// TIA Portal V19 program export: 6 tag tables, 0 data types, 4 data blocks, 10 code blocks (in call order from the OBs), 11 instance data blocks

VAR_GLOBAL   // PLC tag table "Default tag table"
   RETVAL_WWW AT %MW80 : Int;
   LampeStart AT %Q1.0 : Bool;
   Start_Stop AT %M10.0 : Bool;
   Compteur AT %MW2 : Int;
   PieceMax AT %MW100 : Int;
   "Compteur Bonnes Pièces" AT %MW10 : Int;
   "Compteur Mauvaises Pièces" AT %MW12 : Int;
   "Pointeur 1" AT %MD50 : DWord;
   "Pointeur 2" AT %MD54 : DWord;
   "A CHANGER" AT %MW200 : Word;
END_VAR

VAR_GLOBAL   // PLC tag table "Entrées"
   PART_AV AT %I0.0 : Bool;   // Détection pièce disponible
   B2 AT %I0.1 : Bool;   // Détection pièces (pas noir)
   B4 AT %I0.2 : Bool;   // Barrière sécurité
   "1B1" AT %I0.4 : Bool;   // Vérin 1A1 position haute
   "1B2" AT %I0.5 : Bool;   // Vérin 1A1 position basse
   "2B1" AT %I0.6 : Bool;   // Vérin 2A1 rentré
   Start AT %I1.0 : Bool;   // Départ cycle
   Stop AT %I1.1 : Bool;   // Fin cycle
   Reset AT %I1.3 : Bool;   // Initialisation station
   Analogique AT %IW800 : Int;   // Capteur analogique
END_VAR

VAR_GLOBAL   // PLC tag table "Mémoires"
   "Hauteur (pourcentage)" AT %MD0 : Real;   // Valeur de la hauteur de la pièce en pourcentage
   "Activer Q1" AT %M4.0 : Bool;   // Mémoire pour activer Q1
   "Mémoire compteur noires" AT %M4.1 : Bool;   // Mémoire pour les fronts montants du cpt noires
   "Mémoire compteur mauvaise hauteur" AT %M4.2 : Bool;   // Mémoire pour les fronts montants du cpt mauvaises pièces
   "Mémoire compteur bonne hauteur" AT %M4.3 : Bool;   // Mémoire pour les fronts montants du cpt bonnes pièces
   "Clock 1Hz" AT %M250.5 : Bool;
   "Clock 2Hz" AT %M250.3 : Bool;
   "Clock 0,625Hz" AT %M250.6 : Bool;
   "Clock 0,5Hz" AT %M250.7 : Bool;
   "Clock 1,5Hz" AT %M250.4 : Bool;
   "Clock 2,5Hz" AT %M250.2 : Bool;
   "Clock 5Hz" AT %M250.1 : Bool;
   "Clock 10Hz" AT %M250.0 : Bool;
   RETVAL_WWW AT %MW80 : Int;
   Start_Stop AT %M10.0 : Bool;
   Compteur AT %MW2 : Int;
   PieceMax AT %MW100 : Int;
   "Compteur Bonnes Pièces" AT %MW10 : Int;
   "Compteur Mauvaises Pièces" AT %MW12 : Int;
   "Pointeur 1" AT %MD50 : DWord;
   "Pointeur 2" AT %MD54 : DWord;
   "A CHANGER" AT %MW200 : Word;
   "NB Bonnes Pièces" AT %MW26 : Word;   // Nombre des bonnes pièces à afficher sur le web serveur
   "NB Mauvaises Pièces" AT %MW28 : Word;   // Nombre des mauvaises pièces à afficher sur le web serveur
END_VAR

VAR_GLOBAL   // PLC tag table "Sorties"
   "1M2" AT %Q0.0 : Bool;   // Descente vérin élévation pièce
   "1M1" AT %Q0.1 : Bool;   // Montée vérin élévation pièce
   "2M1" AT %Q0.2 : Bool;   // Sortie vérin éjection pièce
   "3M1" AT %Q0.3 : Bool;   // Activation toboggan pneumatique
   LStart AT %Q1.0 : Bool;   // Lampe BP Start
   LReset AT %Q1.1 : Bool;   // Lampe BP Reset
   Q1 AT %Q1.2 : Bool;   // Voyant lumineux Q1
   Q2 AT %Q1.3 : Bool;   // Voyant lumineux Q2
END_VAR

VAR_GLOBAL   // PLC tag table "Test - Copy"
   test1 AT %M120.0 : Bool;
   test2 AT %M120.1 : Bool;
END_VAR

VAR_GLOBAL   // PLC tag table "Test"
   test1 AT %M120.0 : Bool;
   test2 AT %M120.1 : Bool;
END_VAR

DATA_BLOCK "DB Bonnes Pièces"   // DB14
// stored: AutoNumber false
   VAR RETAIN
      "Nb_J-1" : Int;
      "Nb_J-2" : Int;
      "Nb_J-3" : Int;
      "Nb_J-4" : Int;
      "Nb_J-5" : Int;
      "Nb_J-6" : Int;
      "Nb_J-7" : Int;
      "Nb_J-8" : Int;
      "Nb_J-9" : Int;
      "Nb_J-10" : Int;
      "Nb_J-11" : Int;
      "Nb_J-12" : Int;
      "Nb_J-13" : Int;
      "Nb_J-14" : Int;
      "Nb_J-15" : Int;
      "Nb_J-16" : Int;
      "Nb_J-17" : Int;
      "Nb_J-18" : Int;
      "Nb_J-19" : Int;
      "Nb_J-20" : Int;
      "Nb_J-21" : Int;
      "Nb_J-22" : Int;
      "Nb_J-23" : Int;
      "Nb_J-24" : Int;
      "Nb_J-25" : Int;
      "Nb_J-26" : Int;
      "Nb_J-27" : Int;
      "Nb_J-28" : Int;
      "Nb_J-29" : Int;
      "Nb_J-30" : Int;
      "Nb_J-31" : Int;
   END_VAR
BEGIN
END_DATA_BLOCK

DATA_BLOCK "DB Mauvaises Pièces"   // DB13
// stored: AutoNumber false
   VAR RETAIN
      "Nb_J-1" : Int;
      "Nb_J-2" : Int;
      "Nb_J-3" : Int;
      "Nb_J-4" : Int;
      "Nb_J-5" : Int;
      "Nb_J-6" : Int;
      "Nb_J-7" : Int;
      "Nb_J-8" : Int;
      "Nb_J-9" : Int;
      "Nb_J-10" : Int;
      "Nb_J-11" : Int;
      "Nb_J-12" : Int;
      "Nb_J-13" : Int;
      "Nb_J-14" : Int;
      "Nb_J-15" : Int;
      "Nb_J-16" : Int;
      "Nb_J-17" : Int;
      "Nb_J-18" : Int;
      "Nb_J-19" : Int;
      "Nb_J-20" : Int;
      "Nb_J-21" : Int;
      "Nb_J-22" : Int;
      "Nb_J-23" : Int;
      "Nb_J-24" : Int;
      "Nb_J-25" : Int;
      "Nb_J-26" : Int;
      "Nb_J-27" : Int;
      "Nb_J-28" : Int;
      "Nb_J-29" : Int;
      "Nb_J-30" : Int;
      "Nb_J-31" : Int;
   END_VAR
BEGIN
END_DATA_BLOCK

DATA_BLOCK "Grosse data"   // DB1
   VAR RETAIN
      "Grosse donnée" : Bool;
      "Une autre grosse donnée" : Int;
   END_VAR
BEGIN
END_DATA_BLOCK

DATA_BLOCK "Mémoires"   // DB2
   VAR RETAIN
      "Mode Manuel" : Bool;
      "Affichage hauteur" : Int;
      "HMI BP Ascenceur Haut" : Bool;
      "HMI BP Ascenceur Bas" : Bool;
      "HMI BP Ejection" : Bool;
      "HMI SW Glissière" : Bool;
      "Erreur Montée Ascenceur" : Int;
      "Erreur Descente Ascenceur" : Int;
      "Erreur Ejection" : Int;
      "Erreur Capteurs" : Int;
   END_VAR
BEGIN
END_DATA_BLOCK

ORGANIZATION_BLOCK "Main"   // OB1, LAD, ProgramCycle
TITLE = "Main Program Sweep (Cycle)"
   VAR_TEMP
      OB1_EV_CLASS : Byte;   // Bits 0-3 = 1 (Coming event), Bits 4-7 = 1 (Event class 1)
      OB1_SCAN_1 : Byte;   // 1 (Cold restart scan 1 of OB 1), 3 (Scan 2-n of OB 1)
      OB1_PRIORITY : Byte;   // Priority of OB Execution
      OB1_OB_NUMBR : Byte;   // 1 (Organization block 1, OB1)
      OB1_RESERVED_1 : Byte;   // Reserved for system
      OB1_RESERVED_2 : Byte;   // Reserved for system
      OB1_PREV_CYCLE : Int;   // Cycle time of previous OB1 scan (milliseconds)
      OB1_MIN_CYCLE : Int;   // Minimum cycle time of OB1 (milliseconds)
      OB1_MAX_CYCLE : Int;   // Maximum cycle time of OB1 (milliseconds)
      OB1_DATE_TIME : Date_And_Time;   // Date and time OB1 started
   END_VAR
BEGIN

REGION Network 1
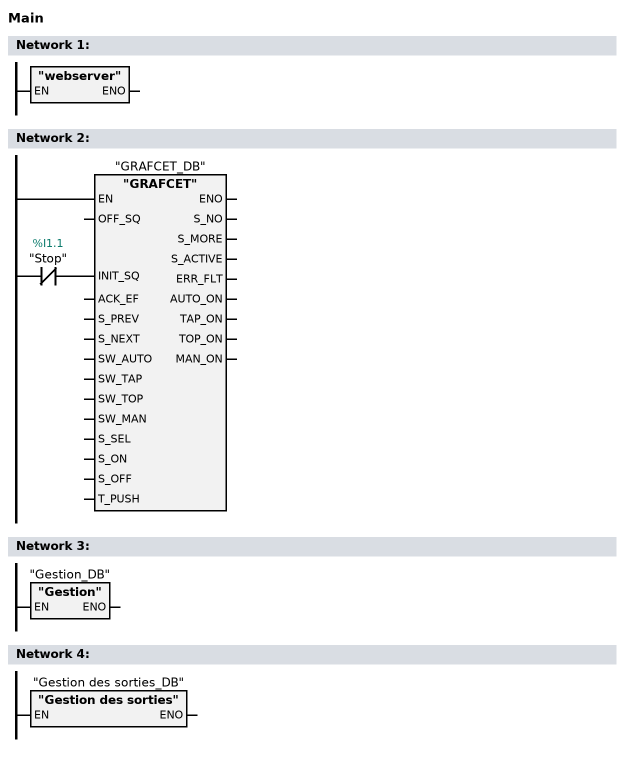
   RUNG wire#powerrail
      "webserver"()
   END_RUNG
   // the same network as SCL:
   "webserver"();
END_REGION

REGION Network 2
   RUNG wire#powerrail
      "GRAFCET_DB"(INIT_SQ := wire#w1, OFF_SQ :=, ACK_EF :=, S_PREV :=, S_NEXT :=, SW_AUTO :=, SW_TAP :=, SW_TOP :=, SW_MAN :=, S_SEL :=, S_ON :=, S_OFF :=, T_PUSH :=, S_NO =>, S_MORE =>, S_ACTIVE =>, ERR_FLT =>, AUTO_ON =>, TAP_ON =>, TOP_ON =>, MAN_ON =>)
   END_RUNG
   RUNG wire#powerrail
      I_Contact( "Stop" )
   END_RUNG wire#w1
   // the same network as SCL:
   "GRAFCET_DB"(INIT_SQ := NOT "Stop");   // "GRAFCET"
END_REGION

REGION Network 3
   RUNG wire#powerrail
      "Gestion_DB"()
   END_RUNG
   // the same network as SCL:
   "Gestion_DB"();   // "Gestion"
END_REGION

REGION Network 4
   RUNG wire#powerrail
      "Gestion des sorties_DB"()
   END_RUNG
   // the same network as SCL:
   "Gestion des sorties_DB"();   // "Gestion des sorties"
END_REGION

NETWORK
TITLE = Call system diagnostics block
      CALL  "RSE_FB", "RSE_DB";
END_ORGANIZATION_BLOCK

FUNCTION "webserver" : Void   // FC1, LAD
   VAR_TEMP
      RET_VAL_1 : Int;
   END_VAR
BEGIN

REGION Network 1
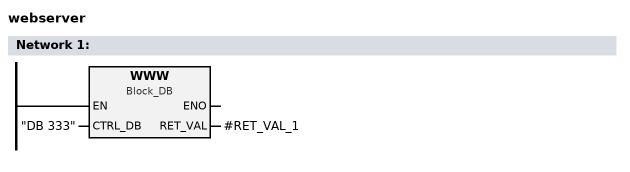
   RUNG wire#powerrail
      { S7_Templates := "value_type := Block_DB" } WWW(CTRL_DB := "DB 333", RET_VAL => #RET_VAL_1)
   END_RUNG
   // the same network as SCL:
   #RET_VAL_1 := WWW(CTRL_DB := "DB 333");
END_REGION
END_FUNCTION

FUNCTION_BLOCK "GRAFCET"   // FB1, GRAPH
   VAR_INPUT
      OFF_SQ { ExternalAccessible := 'False'; ExternalVisible := 'False'; ExternalWritable := 'False'} : Bool := false;   // Turn sequence off
      INIT_SQ { ExternalAccessible := 'False'; ExternalVisible := 'False'; ExternalWritable := 'False'} : Bool := false;   // Set sequence to initial state
      ACK_EF { ExternalAccessible := 'False'; ExternalVisible := 'False'; ExternalWritable := 'False'} : Bool := false;   // Acknowledge all errors and faults
      S_PREV { ExternalAccessible := 'False'; ExternalVisible := 'False'; ExternalWritable := 'False'} : Bool := false;   // Output previous step in parameter S_NO
      S_NEXT { ExternalAccessible := 'False'; ExternalVisible := 'False'; ExternalWritable := 'False'} : Bool := false;   // Indicate next step in parameter S_NO
      SW_AUTO { ExternalAccessible := 'False'; ExternalVisible := 'False'; ExternalWritable := 'False'} : Bool := false;   // Automatic mode
      SW_TAP { ExternalAccessible := 'False'; ExternalVisible := 'False'; ExternalWritable := 'False'} : Bool := false;   // Semiautomatic/switch with transition
      SW_TOP { ExternalAccessible := 'False'; ExternalVisible := 'False'; ExternalWritable := 'False'} : Bool := false;   // Semiautomatic/ignore transition
      SW_MAN { ExternalAccessible := 'False'; ExternalVisible := 'False'; ExternalWritable := 'False'} : Bool := false;   // Manual mode
      S_SEL { ExternalAccessible := 'False'; ExternalVisible := 'False'; ExternalWritable := 'False'} : Int := 0;   // Select step to be output to S_NO
      S_ON { ExternalAccessible := 'False'; ExternalVisible := 'False'; ExternalWritable := 'False'} : Bool := false;   // Activate step indicated in S_NO
      S_OFF { ExternalAccessible := 'False'; ExternalVisible := 'False'; ExternalWritable := 'False'} : Bool := false;   // Deactivate step indicated S_NO
      T_PUSH { ExternalAccessible := 'False'; ExternalVisible := 'False'; ExternalWritable := 'False'} : Bool := false;   // Enable transition to switch in semi automatic mode
   END_VAR
   VAR_OUTPUT
      S_NO { ExternalAccessible := 'False'; ExternalVisible := 'False'; ExternalWritable := 'False'} : Int := 0;   // Step number
      S_MORE { ExternalAccessible := 'False'; ExternalVisible := 'False'; ExternalWritable := 'False'} : Bool := false;   // More steps are available and can be shown in S_NO
      S_ACTIVE { ExternalAccessible := 'False'; ExternalVisible := 'False'; ExternalWritable := 'False'} : Bool := false;   // Step indicated in S_NO is active
      ERR_FLT { ExternalAccessible := 'False'; ExternalVisible := 'False'; ExternalWritable := 'False'} : Bool := false;   // Interlock or supervision group error
      AUTO_ON { ExternalAccessible := 'False'; ExternalVisible := 'False'; ExternalWritable := 'False'} : Bool := false;   // Automatic mode is active
      TAP_ON { ExternalAccessible := 'False'; ExternalVisible := 'False'; ExternalWritable := 'False'} : Bool := false;   // Semiautomatic mode/step with transition enabled
      TOP_ON { ExternalAccessible := 'False'; ExternalVisible := 'False'; ExternalWritable := 'False'} : Bool := false;   // Semiautomatic mode/ignore transition enabled
      MAN_ON { ExternalAccessible := 'False'; ExternalVisible := 'False'; ExternalWritable := 'False'} : Bool := false;   // Manual mode is active
   END_VAR
   VAR
      S_DISPLAY { ExternalAccessible := 'False'; ExternalVisible := 'False'; ExternalWritable := 'False'} : Int;   // Internal display of output parameter S_NO
      S_SEL_OLD { ExternalAccessible := 'False'; ExternalVisible := 'False'; ExternalWritable := 'False'} : Int;   // Previous value in S_SEL
      S_DISPIDX { ExternalAccessible := 'False'; ExternalVisible := 'False'; ExternalWritable := 'False'} : Byte;   // Index of the step in S_NO
      T_DISPIDX { ExternalAccessible := 'False'; ExternalVisible := 'False'; ExternalWritable := 'False'} : Byte;   // Index of the transition displayed in T_NO
      MOP { ExternalAccessible := 'False'; ExternalVisible := 'False'; ExternalWritable := 'False'} : Struct   // Mode
         AUTO : Bool := true;   // Status: automatic mode
         MAN : Bool := false;   // Status: manual mode
         TAP : Bool := false;   // Status: semi automatic/switch with transition
         TOP : Bool := false;   // Status: semi automatic/ignore transition
         ACK_S : Bool := false;   // Request: acknowledge step at parameter S_NO
         REG_S : Bool := false;   // Request: register step indicated in S_NO
         T_PREV : Bool := false;   // Request: output previous valid transition in T_NO
         T_NEXT : Bool := false;   // Request: output next valid transition in T_NO
         LOCK : Bool := true;   // Status: interlocks activated
         SUP : Bool := true;   // Status: supervisions activated
         ACKREQ : Bool := true;   // Status: acknowledgment required
         SSKIP : Bool := false;   // Status: "Skip steps" enabled
         OFF : Bool := false;   // Request: deactivate all steps
         INIT : Bool := true;   // Request: set sequence to initial state
         HALT : Bool := false;   // Status: sequence halted
         TMS_HALT : Bool := false;   // Status: all internal timers held
         OPS_ZERO : Bool := false;   // Status: set all operands processed with N, L, D instructions to 0
         SACT_DISP : Bool := true;   // Status: display active steps only
         SEF_DISP : Bool := false;   // Status: display only steps with errors and disrupted steps
         SALL_DISP : Bool := false;   // Status: display all steps
         S_PREV : Bool := false;   // Request: output previous step to S_NO
         S_NEXT : Bool := false;   // Request: Output next step at S_NO parameter
         S_SELOK : Bool := false;   // Request: output step number from S_SEL to S_NO
         S_ON : Bool := false;   // Request: activate step indicated in S_NO
         S_OFF : Bool := false;   // Request: deactivate step at parameter S_NO
         T_PUSH : Bool := false;   // Request: transition switching enabled
         REG : Bool := false;   // Request: register all interlock and supervision errors
         ACK : Bool := false;   // Request: acknowledge all interlock and supervision errors
         IL_PERM : Bool := false;   // Status: permanent processing of all interlocks
         T_PERM : Bool := false;   // Status: permanent processing of all transitions
         ILP_MAN : Bool := false;   // Status: permanent processing of all interlocks in manual mode
      END_STRUCT;
      TICKS { ExternalAccessible := 'False'; ExternalVisible := 'False'; ExternalWritable := 'False'} : Struct   // Clock speeds
         DELTA : Time := T#0ms;   // Time difference between cycles
         OLD : Time := T#0ms;   // 10 ms clock counter value in last cycle
         NEW : Time := T#0ms;   // 10 ms clock counter value in this cycle
      END_STRUCT;
      SQ_FLAGS { ExternalAccessible := 'False'; ExternalVisible := 'False'; ExternalWritable := 'False'} : Struct   // Sequence bit memory
         ERR_FLT : Bool := false;   // Interlock and supervision group error
         ERROR : Bool := false;   // Interlock group error
         FAULT : Bool := false;   // Supervision group error
         RT_FAIL : Bool := false;   // Runtime error
         NO_SNO : Bool := false;   // Requested step number not found
         NF_OFL : Bool := false;   // Overflow: too many ON or OFF requests
         SA_OFL : Bool := false;   // Overflow: too many steps active
         TV_OFL : Bool := false;   // Overflow: too many valid transitions
         MSG_OFL : Bool := false;   // Overflow: not enough system resources for ALARM_S
         NO_SWI : Bool := false;   // Do not switch in this cycle
         CYC_OP : Bool := false;   // Cyclic execution of the sequence after initialization
         AS_MSG : Bool := true;   // Alarms during runtime enabled or disabled by instruction
         AS_SEND : Bool := false;   // Send alarms from WR_USMSG or only enter in diagnostics buffer
         SQ_BUSY : Bool := false;   // Internal edge bit memory for sequence processing
         SA_BUSY : Bool := false;   // Internal edge bit memory for sequence processing
         AS_SIG : Bool := false;   // Edge bit memory for alarms from Alarm_S and Alarm_SQ
      END_STRUCT;
   END_VAR
BEGIN
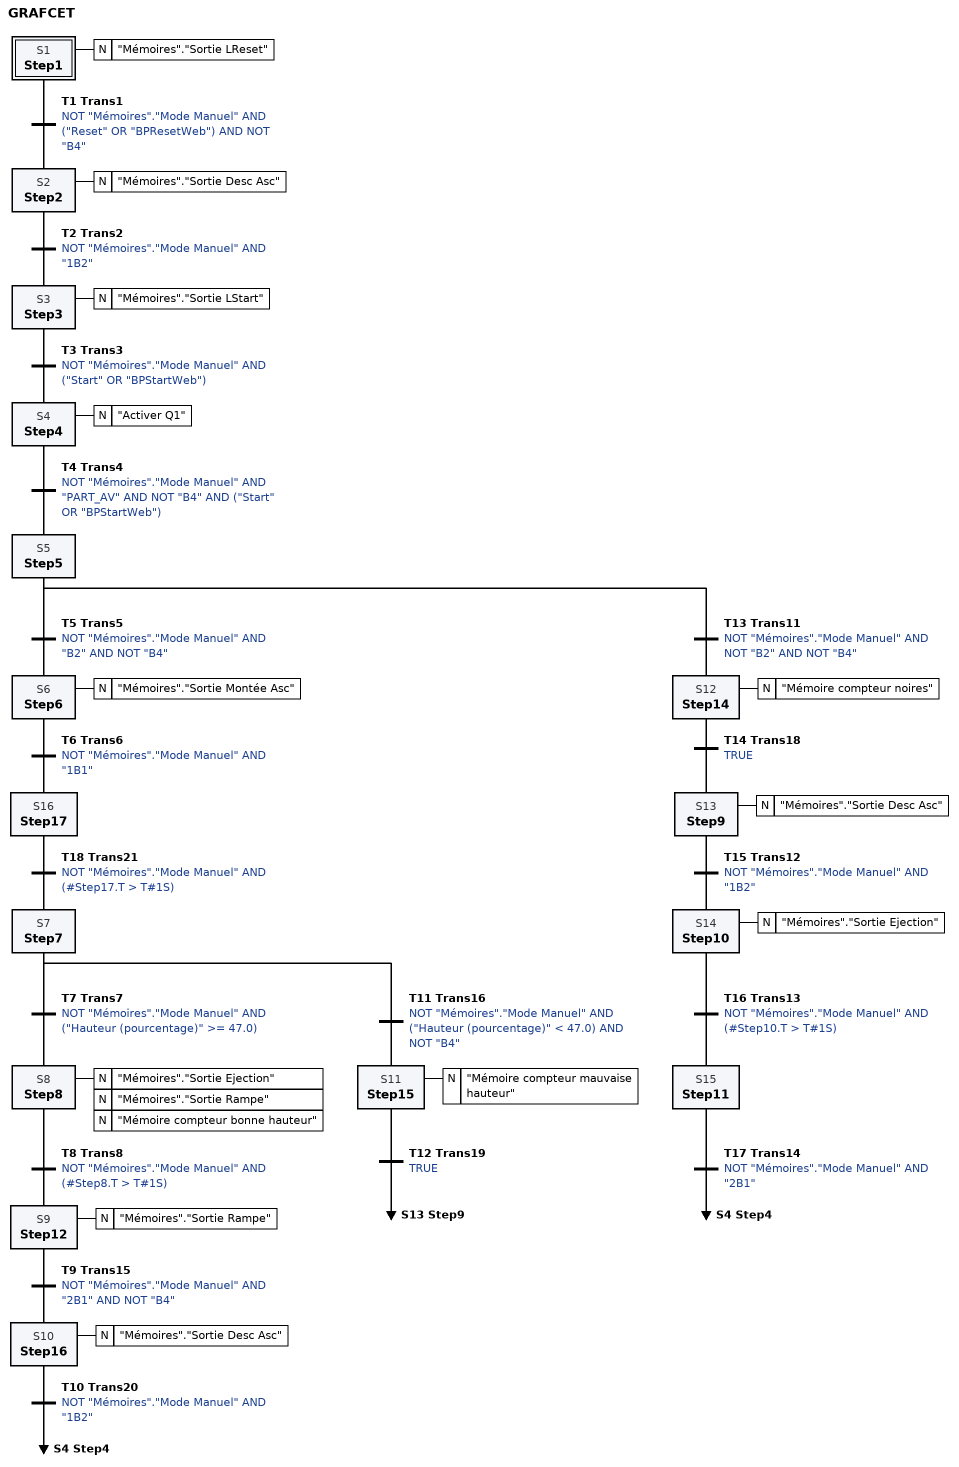
   // sequencer 1: GRAFCET de la séquence de tri
   INITIAL_STEP Step1:   // S1
              N    "Mémoires"."Sortie LReset"
   END_STEP
   TRANSITION Trans1 FROM Step1 TO Step2   // T1
      := NOT "Mémoires"."Mode Manuel" AND ("Reset" OR "BPResetWeb") AND NOT "B4";
   END_TRANSITION
   STEP Step2:   // S2
              N    "Mémoires"."Sortie Desc Asc"
   END_STEP
   TRANSITION Trans2 FROM Step2 TO Step3   // T2
      := NOT "Mémoires"."Mode Manuel" AND "1B2";
   END_TRANSITION
   STEP Step3:   // S3
              N    "Mémoires"."Sortie LStart"
   END_STEP
   TRANSITION Trans3 FROM Step3 TO Step4   // T3
      := NOT "Mémoires"."Mode Manuel" AND ("Start" OR "BPStartWeb");
   END_TRANSITION
   STEP Step4:   // S4
              N    "Activer Q1"
   END_STEP
   TRANSITION Trans4 FROM Step4 TO Step5   // T4
      := NOT "Mémoires"."Mode Manuel" AND "PART_AV" AND NOT "B4" AND ("Start" OR "BPStartWeb");
   END_TRANSITION
   STEP Step5:   // S5
   END_STEP
   TRANSITION Trans5 FROM Step5 TO Step6   // T5
      := NOT "Mémoires"."Mode Manuel" AND "B2" AND NOT "B4";
   END_TRANSITION
   TRANSITION Trans11 FROM Step5 TO Step14   // T13
      := NOT "Mémoires"."Mode Manuel" AND NOT "B2" AND NOT "B4";
   END_TRANSITION
   STEP Step6:   // S6
              N    "Mémoires"."Sortie Montée Asc"
   END_STEP
   TRANSITION Trans6 FROM Step6 TO Step17   // T6
      := NOT "Mémoires"."Mode Manuel" AND "1B1";
   END_TRANSITION
   STEP Step7:   // S7
   END_STEP
   TRANSITION Trans7 FROM Step7 TO Step8   // T7
      := NOT "Mémoires"."Mode Manuel" AND ("Hauteur (pourcentage)" >= 47.0);
   END_TRANSITION
   TRANSITION Trans16 FROM Step7 TO Step15   // T11
      := NOT "Mémoires"."Mode Manuel" AND ("Hauteur (pourcentage)" < 47.0) AND NOT "B4";
   END_TRANSITION
   STEP Step8:   // S8
              N    "Mémoires"."Sortie Ejection"
              N    "Mémoires"."Sortie Rampe"
              N    "Mémoire compteur bonne hauteur"
   END_STEP
   TRANSITION Trans8 FROM Step8 TO Step12   // T8
      := NOT "Mémoires"."Mode Manuel" AND (#Step8.T > T#1S);
   END_TRANSITION
   STEP Step9:   // S13
              N    "Mémoires"."Sortie Desc Asc"
   END_STEP
   TRANSITION Trans12 FROM Step9 TO Step10   // T15
      := NOT "Mémoires"."Mode Manuel" AND "1B2";
   END_TRANSITION
   STEP Step10:   // S14
              N    "Mémoires"."Sortie Ejection"
   END_STEP
   TRANSITION Trans13 FROM Step10 TO Step11   // T16
      := NOT "Mémoires"."Mode Manuel" AND (#Step10.T > T#1S);
   END_TRANSITION
   STEP Step11:   // S15
   END_STEP
   TRANSITION Trans14 FROM Step11 TO Step4   // T17, jump
      := NOT "Mémoires"."Mode Manuel" AND "2B1";
   END_TRANSITION
   STEP Step12:   // S9
              N    "Mémoires"."Sortie Rampe"
   END_STEP
   TRANSITION Trans15 FROM Step12 TO Step16   // T9
      := NOT "Mémoires"."Mode Manuel" AND "2B1" AND NOT "B4";
   END_TRANSITION
   STEP Step14:   // S12
              N    "Mémoire compteur noires"
   END_STEP
   TRANSITION Trans18 FROM Step14 TO Step9   // T14
      := TRUE;
   END_TRANSITION
   STEP Step15:   // S11
              N    "Mémoire compteur mauvaise hauteur"
   END_STEP
   TRANSITION Trans19 FROM Step15 TO Step9   // T12, jump
      := TRUE;
   END_TRANSITION
   STEP Step16:   // S10
              N    "Mémoires"."Sortie Desc Asc"
   END_STEP
   TRANSITION Trans20 FROM Step16 TO Step4   // T10, jump
      := NOT "Mémoires"."Mode Manuel" AND "1B2";
   END_TRANSITION
   STEP Step17:   // S16
   END_STEP
   TRANSITION Trans21 FROM Step17 TO Step7   // T18
      := NOT "Mémoires"."Mode Manuel" AND (#Step17.T > T#1S);
   END_TRANSITION
END_FUNCTION_BLOCK

FUNCTION_BLOCK "Gestion"   // FB2, LAD
   VAR
      "Code erreur" : Word;
      "FM Noires" : Bool;
      "FM Mauvaises" : Bool;
      "FM Bonnes" : Bool;
   END_VAR
   VAR_TEMP   // added for the SCL form of the ladder/FBD networks
      _w1 : Bool;
   END_VAR
BEGIN

REGION Network 1: Scale de la valeur d'entrée analogique
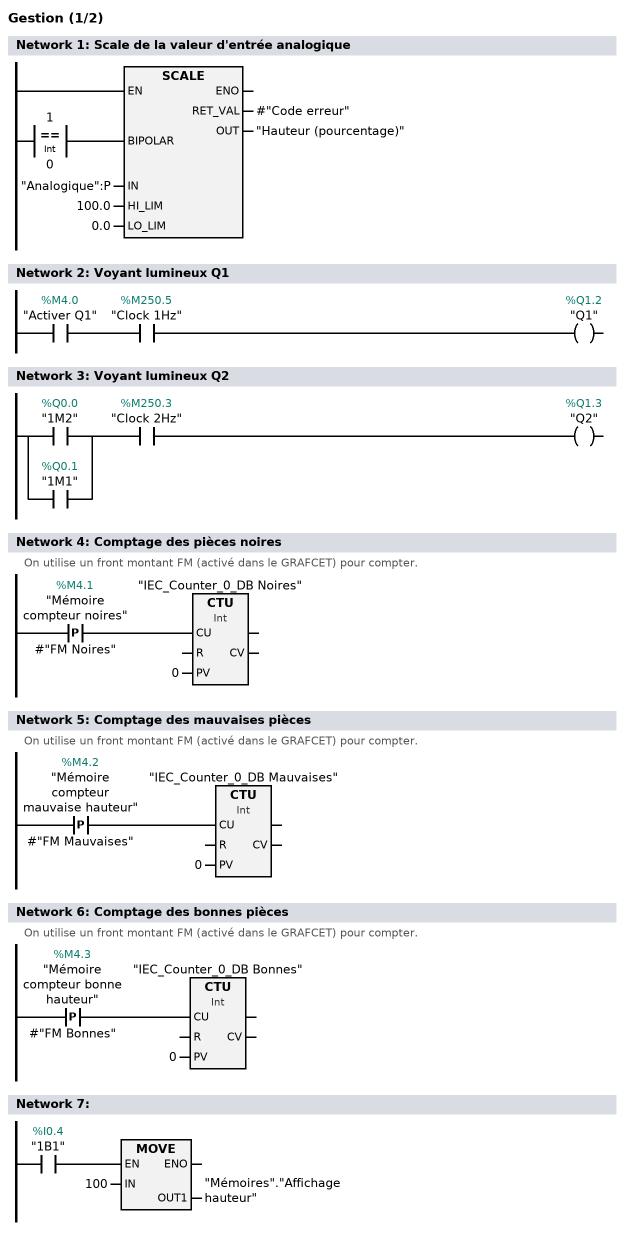
   #"Code erreur" := SCALE(BIPOLAR := 1 = 0,
                           IN := "Analogique":P,
                           HI_LIM := 100.0,
                           LO_LIM := 0.0,
                           OUT => "Hauteur (pourcentage)");
END_REGION

REGION Network 2: Voyant lumineux Q1
   RUNG wire#powerrail
      Contact( "Activer Q1" )
      Contact( "Clock 1Hz" )
      Coil( "Q1" )
   END_RUNG
   // the same network as SCL:
   "Q1" := "Activer Q1" AND "Clock 1Hz";
END_REGION

REGION Network 3: Voyant lumineux Q2
   RUNG wire#powerrail
      Contact( "1M2" )
      wire#w1
      Contact( "Clock 2Hz" )
      Coil( "Q2" )
   END_RUNG
   RUNG wire#powerrail
      Contact( "1M1" )
   END_RUNG wire#w1
   // the same network as SCL:
   "Q2" := ("1M2" OR "1M1") AND "Clock 2Hz";
END_REGION

REGION Network 4: Comptage des pièces noires
   // On utilise un front montant FM (activé dans le GRAFCET) pour compter.
   RUNG wire#powerrail
      P_Contact(operand := "Mémoire compteur noires", bit := #"FM Noires")
      { S7_Templates := "value_type := Int" } "IEC_Counter_0_DB Noires".CTU(r :=, pv := 0, cv =>)
   END_RUNG
   // the same network as SCL:
   #_w1 := "Mémoire compteur noires" AND NOT #"FM Noires";   // rising edge of "Mémoire compteur noires"
   #"FM Noires" := "Mémoire compteur noires";
   "IEC_Counter_0_DB Noires".CTU(CU := #_w1, PV := 0);
END_REGION

REGION Network 5: Comptage des mauvaises pièces
   // On utilise un front montant FM (activé dans le GRAFCET) pour compter.
   RUNG wire#powerrail
      P_Contact(operand := "Mémoire compteur mauvaise hauteur", bit := #"FM Mauvaises")
      { S7_Templates := "value_type := Int" } "IEC_Counter_0_DB Mauvaises".CTU(r :=, pv := 0, cv =>)
   END_RUNG
   // the same network as SCL:
   #_w1 := "Mémoire compteur mauvaise hauteur" AND NOT #"FM Mauvaises";   // rising edge of "Mémoire compteur mauvaise hauteur"
   #"FM Mauvaises" := "Mémoire compteur mauvaise hauteur";
   "IEC_Counter_0_DB Mauvaises".CTU(CU := #_w1, PV := 0);
END_REGION

REGION Network 6: Comptage des bonnes pièces
   // On utilise un front montant FM (activé dans le GRAFCET) pour compter.
   RUNG wire#powerrail
      P_Contact(operand := "Mémoire compteur bonne hauteur", bit := #"FM Bonnes")
      { S7_Templates := "value_type := Int" } "IEC_Counter_0_DB Bonnes".CTU(r :=, pv := 0, cv =>)
   END_RUNG
   // the same network as SCL:
   #_w1 := "Mémoire compteur bonne hauteur" AND NOT #"FM Bonnes";   // rising edge of "Mémoire compteur bonne hauteur"
   #"FM Bonnes" := "Mémoire compteur bonne hauteur";
   "IEC_Counter_0_DB Bonnes".CTU(CU := #_w1, PV := 0);
END_REGION

REGION Network 7
   RUNG wire#powerrail
      Contact( "1B1" )
      { S7_GenerateENO := "TRUE" } Move(in := 100, out1 => "Mémoires"."Affichage hauteur")
   END_RUNG
   // the same network as SCL:
   IF "1B1" THEN "Mémoires"."Affichage hauteur" := 100; END_IF;
END_REGION

REGION Network 8
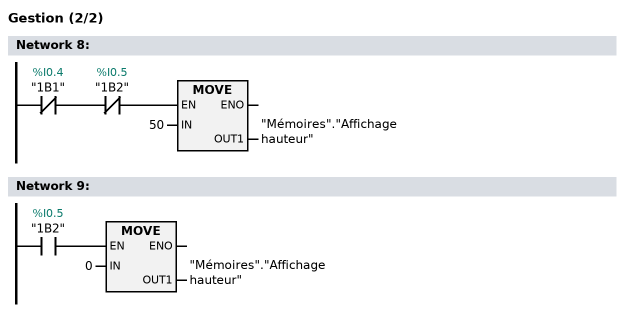
   RUNG wire#powerrail
      I_Contact( "1B1" )
      I_Contact( "1B2" )
      { S7_GenerateENO := "TRUE" } Move(in := 50, out1 => "Mémoires"."Affichage hauteur")
   END_RUNG
   // the same network as SCL:
   IF NOT "1B1" AND NOT "1B2" THEN "Mémoires"."Affichage hauteur" := 50; END_IF;
END_REGION

REGION Network 9
   RUNG wire#powerrail
      Contact( "1B2" )
      { S7_GenerateENO := "TRUE" } Move(in := 0, out1 => "Mémoires"."Affichage hauteur")
   END_RUNG
   // the same network as SCL:
   IF "1B2" THEN "Mémoires"."Affichage hauteur" := 0; END_IF;
END_REGION
END_FUNCTION_BLOCK

FUNCTION_BLOCK "Gestion des sorties"   // FB3, LAD
BEGIN

REGION Network 1: Descente vérin élévation pièce
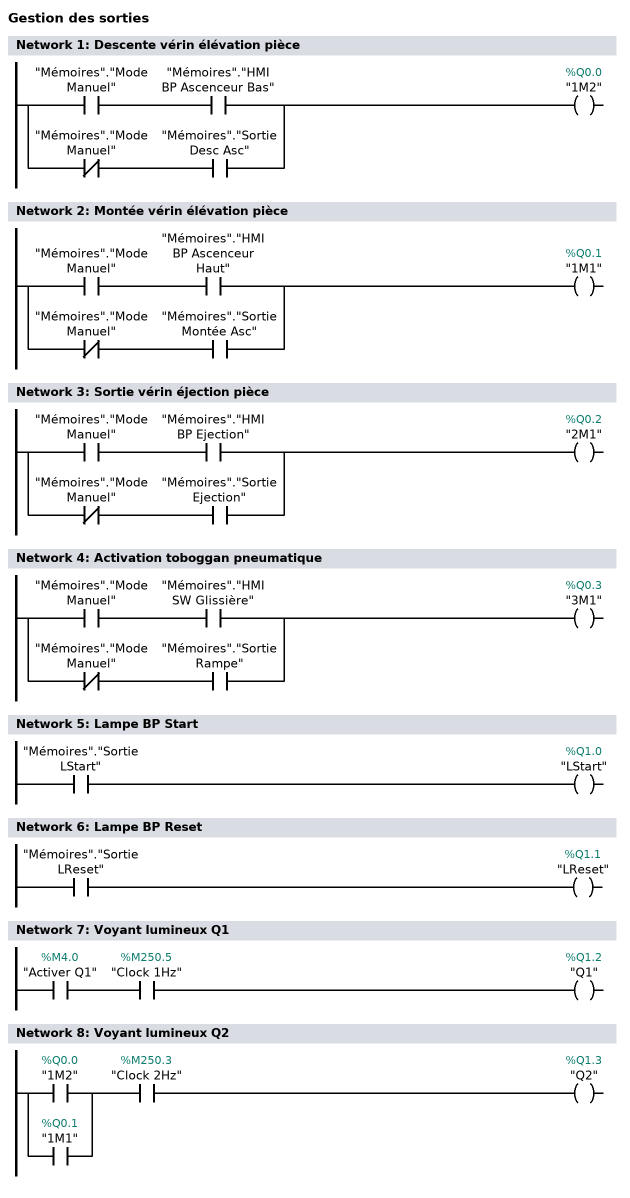
   RUNG wire#powerrail
      Contact( "Mémoires"."Mode Manuel" )
      Contact( "Mémoires"."HMI BP Ascenceur Bas" )
      wire#w1
      Coil( "1M2" )
   END_RUNG
   RUNG wire#powerrail
      I_Contact( "Mémoires"."Mode Manuel" )
      Contact( "Mémoires"."Sortie Desc Asc" )
   END_RUNG wire#w1
   // the same network as SCL:
   "1M2" := ("Mémoires"."Mode Manuel" AND "Mémoires"."HMI BP Ascenceur Bas") OR (NOT "Mémoires"."Mode Manuel" AND "Mémoires"."Sortie Desc Asc");
END_REGION

REGION Network 2: Montée vérin élévation pièce
   RUNG wire#powerrail
      Contact( "Mémoires"."Mode Manuel" )
      Contact( "Mémoires"."HMI BP Ascenceur Haut" )
      wire#w1
      Coil( "1M1" )
   END_RUNG
   RUNG wire#powerrail
      I_Contact( "Mémoires"."Mode Manuel" )
      Contact( "Mémoires"."Sortie Montée Asc" )
   END_RUNG wire#w1
   // the same network as SCL:
   "1M1" := ("Mémoires"."Mode Manuel" AND "Mémoires"."HMI BP Ascenceur Haut") OR (NOT "Mémoires"."Mode Manuel" AND "Mémoires"."Sortie Montée Asc");
END_REGION

REGION Network 3: Sortie vérin éjection pièce
   RUNG wire#powerrail
      Contact( "Mémoires"."Mode Manuel" )
      Contact( "Mémoires"."HMI BP Ejection" )
      wire#w1
      Coil( "2M1" )
   END_RUNG
   RUNG wire#powerrail
      I_Contact( "Mémoires"."Mode Manuel" )
      Contact( "Mémoires"."Sortie Ejection" )
   END_RUNG wire#w1
   // the same network as SCL:
   "2M1" := ("Mémoires"."Mode Manuel" AND "Mémoires"."HMI BP Ejection") OR (NOT "Mémoires"."Mode Manuel" AND "Mémoires"."Sortie Ejection");
END_REGION

REGION Network 4: Activation toboggan pneumatique
   RUNG wire#powerrail
      Contact( "Mémoires"."Mode Manuel" )
      Contact( "Mémoires"."HMI SW Glissière" )
      wire#w1
      Coil( "3M1" )
   END_RUNG
   RUNG wire#powerrail
      I_Contact( "Mémoires"."Mode Manuel" )
      Contact( "Mémoires"."Sortie Rampe" )
   END_RUNG wire#w1
   // the same network as SCL:
   "3M1" := ("Mémoires"."Mode Manuel" AND "Mémoires"."HMI SW Glissière") OR (NOT "Mémoires"."Mode Manuel" AND "Mémoires"."Sortie Rampe");
END_REGION

REGION Network 5: Lampe BP Start
   RUNG wire#powerrail
      Contact( "Mémoires"."Sortie LStart" )
      Coil( "LStart" )
   END_RUNG
   // the same network as SCL:
   "LStart" := "Mémoires"."Sortie LStart";
END_REGION

REGION Network 6: Lampe BP Reset
   RUNG wire#powerrail
      Contact( "Mémoires"."Sortie LReset" )
      Coil( "LReset" )
   END_RUNG
   // the same network as SCL:
   "LReset" := "Mémoires"."Sortie LReset";
END_REGION

REGION Network 7: Voyant lumineux Q1
   RUNG wire#powerrail
      Contact( "Activer Q1" )
      Contact( "Clock 1Hz" )
      Coil( "Q1" )
   END_RUNG
   // the same network as SCL:
   "Q1" := "Activer Q1" AND "Clock 1Hz";
END_REGION

REGION Network 8: Voyant lumineux Q2
   RUNG wire#powerrail
      Contact( "1M2" )
      wire#w1
      Contact( "Clock 2Hz" )
      Coil( "Q2" )
   END_RUNG
   RUNG wire#powerrail
      Contact( "1M1" )
   END_RUNG wire#w1
   // the same network as SCL:
   "Q2" := ("1M2" OR "1M1") AND "Clock 2Hz";
END_REGION
END_FUNCTION_BLOCK

ORGANIZATION_BLOCK "OBNL_FLT"   // OB85, STL, AccessError
TITLE = "Organization Block (OB) Not Loaded Fault"
   VAR_TEMP
      OB85_EV_CLASS : Byte;   // 16#35 Event class 3
      OB85_FLT_ID : Byte;   // 16#XX, Fault identification code
      OB85_PRIORITY : Byte;   // Priority of OB Execution
      OB85_OB_NUMBR : Byte;   // 85 (Organization block 85, OB85)
      OB85_RESERVED_1 : Byte;   // Reserved for system
      OB85_RESERVED_2 : Byte;   // Reserved for system
      OB85_RESERVED_3 : Int;   // Reserved for system
      OB85_ERR_EV_CLASS : Byte;   // Class of event causing error
      OB85_ERR_EV_NUM : Byte;   // Number of event causing error
      OB85_OB_PRIOR : Byte;   // Priority of OB causing error
      OB85_OB_NUM : Byte;   // Number of OB causing error
      OB85_DATE_TIME : Date_And_Time;   // Date and time OB85 started
   END_VAR
BEGIN

NETWORK
TITLE = 
      L     b#16#A1;  //
      L     #OB85_FLT_ID;
      ==I;
      JC    K_OB;
      L     b#16#A2;  //
      ==I;
      JC    K_OB;
      L     b#16#A3;  //
      L     #OB85_FLT_ID;
      ==I;
      JC    K_B;
      JU    F_PA;


NETWORK
TITLE = 
K_OB: JU    STOP;
      JU    ENDE;


NETWORK
TITLE = 
K_B:  JU    STOP;
      JU    ENDE;


NETWORK
TITLE = 
F_PA: NOP   0;
      JU    ENDE;


NETWORK
TITLE = 
STOP: CALL  STP;


NETWORK
TITLE = 

//

ENDE: NOP   0;

END_ORGANIZATION_BLOCK

ORGANIZATION_BLOCK "RACK_FLT"   // OB86, STL, RackOrStationFailure
TITLE = "Loss Of Rack Fault"
   VAR_TEMP
      OB86_EV_CLASS : Byte;   // 16#38/39 Event class 3
      OB86_FLT_ID : Byte;   // 16#C1/C4/C5, Fault identification code
      OB86_PRIORITY : Byte;   // Priority of OB Execution
      OB86_OB_NUMBR : Byte;   // 86 (Organization block 86, OB86)
      OB86_RESERVED_1 : Byte;   // Reserved for system
      OB86_RESERVED_2 : Byte;   // Reserved for system
      OB86_MDL_ADDR : Word;   // Base address of IM module in rack with fault
      OB86_RACKS_FLTD : Array[0..31] of Bool;   // Racks in fault
      OB86_DATE_TIME : Date_And_Time;   // Date and time OB86 started
   END_VAR
BEGIN

NETWORK
TITLE = Call system diagnostics block
      CALL  "RSE_FB", "RSE_DB";
END_ORGANIZATION_BLOCK

ORGANIZATION_BLOCK "TOD_INT0"   // OB10, LAD, TimeOfDay
TITLE = "Time of Day Interrupt"
   VAR_TEMP
      OB10_EV_CLASS : Byte;   // Bits 0-3 = 1 (Coming event), Bits 4-7 = 1 (Event class 1)
      OB10_STRT_INFO : Byte;   // 16#11 (OB 10 has started)
      OB10_PRIORITY : Byte;   // Priority of OB Execution
      OB10_OB_NUMBR : Byte;   // 10 (Organization block 10, OB10)
      OB10_RESERVED_1 : Byte;   // Reserved for system
      OB10_RESERVED_2 : Byte;   // Reserved for system
      OB10_PERIOD_EXE : Word;   // Period of execution (once, per minute/hour/day/week/month/year)
      OB10_RESERVED_3 : Int;   // Reserved for system
      OB10_RESERVED_4 : Int;   // Reserved for system
      OB10_DATE_TIME : Date_And_Time;   // Date and time OB10 started
   END_VAR
BEGIN

REGION Network 1
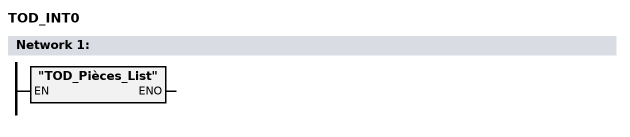
   RUNG wire#powerrail
      "TOD_Pièces_List"()
   END_RUNG
   // the same network as SCL:
   "TOD_Pièces_List"();
END_REGION
END_ORGANIZATION_BLOCK

FUNCTION "TOD_Pièces_List" : Void   // FC2, STL
TITLE = Décalages
// J-1 -> J-2 etc... jusque J-31
BEGIN

NETWORK
TITLE = Décalage Bonnes Pièces
// BONNES PIECES DECALAGE

      OPN   "DB Bonnes Pièces";

//Pointeurs de 2 mémoires qui se suivent
      L     P#58.0;
      T     "Pointeur 1";
      L     P#60.0;
      T     "Pointeur 2";

//Compteur à 30 itérations
      L     30;
bcl1: T     "Compteur Bonnes Pièces";

//transfert JX à JX-1
      L     DBW ["Pointeur 1"];
      T     DBW ["Pointeur 2"];

//On retire 2 car double octet aux pointeurs pour avancer d'un jour
      L     "Pointeur 1";
      L     P#2.0;
      -D;
      T     "Pointeur 1";

      L     "Pointeur 2";
      L     P#2.0;
      -D;
      T     "Pointeur 2";

//Fin de la loop on charge le compteur et le loop enlève 1. Out si =0
      L     "Compteur Bonnes Pièces";
      LOOP  bcl1;


//Ajouter la variable avec Nb pièce de la journée
      L     "A CHANGER";
      T     "DB Bonnes Pièces"."Nb_J-1";

//Nouvelle Journée
      L     0;
      T     "A CHANGER";



NETWORK
TITLE = Décalage Mauvaises Pièces
// PIECES NOIRES DECALAGE

      OPN   "DB Mauvaises Pièces";

//Pointeurs de 2 mémoires qui se suivent
      L     P#58.0;
      T     "Pointeur 1";
      L     P#60.0;
      T     "Pointeur 2";

//Compteur à 30 itérations
      L     30;
bcl2: T     "Compteur Mauvaises Pièces";

//transfert JX à JX-1
      L     DBW ["Pointeur 1"];
      T     DBW ["Pointeur 2"];

//On retire 2 car double octet aux pointeurs pour avancer d'un jour
      L     "Pointeur 1";
      L     P#2.0;
      -D;
      T     "Pointeur 1";

      L     "Pointeur 2";
      L     P#2.0;
      -D;
      T     "Pointeur 2";

//Fin de la loop on charge le compteur et le loop enlève 1. Out si =0
      L     "Compteur Mauvaises Pièces";
      LOOP  bcl2;


//Ajouter la variable avec Nb pièce de la journée
      L     "A CHANGER";
      T     "DB Mauvaises Pièces"."Nb_J-1";

//Nouvelle Journée
      L     0;
      T     "A CHANGER";


END_FUNCTION

FUNCTION "Gros test" : Void   // FC1, LAD
BEGIN

REGION Network 1
   // Voilà un bien gros test...
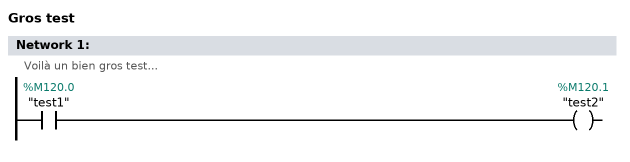
   RUNG wire#powerrail
      Contact( "test1" )
      Coil( "test2" )
   END_RUNG
   // the same network as SCL:
   "test2" := "test1";
END_REGION
END_FUNCTION

DATA_BLOCK "GRAFCET_DB"   // DB6
// stored: InstanceOfName GRAFCET, InstanceOfType FB
"GRAFCET"
BEGIN
END_DATA_BLOCK

DATA_BLOCK "Gestion des sorties MANU_DB"   // DB11
// stored: InstanceOfName Gestion des sorties, InstanceOfType FB
"Gestion des sorties"
BEGIN
END_DATA_BLOCK

DATA_BLOCK "Gestion des sorties_DB"   // DB12
// stored: InstanceOfName Gestion des sorties, InstanceOfType FB
"Gestion des sorties"
BEGIN
END_DATA_BLOCK

DATA_BLOCK "Gestion_DB"   // DB5
// stored: InstanceOfName Gestion, InstanceOfType FB
"Gestion"
BEGIN
END_DATA_BLOCK

DATA_BLOCK "IEC_Timer_0_DB"   // DB7
// stored: InstanceOfName TON_SFB, OfSystemLibElement TON, OfSystemLibVersion 1.0
"TON_SFB"
   // VAR_INPUT
   //    IN : Bool;
   //    PT : Time;
   // END_VAR
   // VAR_OUTPUT
   //    Q : Bool;
   //    ET : Time;
   // END_VAR
   // VAR RETAIN
   //    STATE : Byte;
   //    STIME : Time;
   //    ATIME : Time;
   // END_VAR
BEGIN
END_DATA_BLOCK

DATA_BLOCK "IEC_Timer_0_DB_1"   // DB8
// stored: InstanceOfName TON_SFB, OfSystemLibElement TON, OfSystemLibVersion 1.0
"TON_SFB"
   // VAR_INPUT
   //    IN : Bool;
   //    PT : Time;
   // END_VAR
   // VAR_OUTPUT
   //    Q : Bool;
   //    ET : Time;
   // END_VAR
   // VAR RETAIN
   //    STATE : Byte;
   //    STIME : Time;
   //    ATIME : Time;
   // END_VAR
BEGIN
END_DATA_BLOCK

DATA_BLOCK "IEC_Timer_0_DB_2"   // DB9
// stored: InstanceOfName TON_SFB, OfSystemLibElement TON, OfSystemLibVersion 1.0
"TON_SFB"
   // VAR_INPUT
   //    IN : Bool;
   //    PT : Time;
   // END_VAR
   // VAR_OUTPUT
   //    Q : Bool;
   //    ET : Time;
   // END_VAR
   // VAR RETAIN
   //    STATE : Byte;
   //    STIME : Time;
   //    ATIME : Time;
   // END_VAR
BEGIN
END_DATA_BLOCK

DATA_BLOCK "IEC_Timer_0_DB_3"   // DB10
// stored: InstanceOfName TON_SFB, OfSystemLibElement TON, OfSystemLibVersion 1.0
"TON_SFB"
   // VAR_INPUT
   //    IN : Bool;
   //    PT : Time;
   // END_VAR
   // VAR_OUTPUT
   //    Q : Bool;
   //    ET : Time;
   // END_VAR
   // VAR RETAIN
   //    STATE : Byte;
   //    STIME : Time;
   //    ATIME : Time;
   // END_VAR
BEGIN
END_DATA_BLOCK

DATA_BLOCK "IEC_Counter_0_DB Bonnes"   // DB4
// stored: InstanceOfName CTU_SFB, OfSystemLibElement CTU, OfSystemLibVersion 1.0
"CTU_SFB"
   // VAR_INPUT
   //    CU : Bool;
   //    R : Bool;
   //    PV : Int;
   // END_VAR
   // VAR_OUTPUT
   //    Q : Bool;
   //    CV : Int;
   // END_VAR
   // VAR RETAIN
   //    CUO : Bool;
   // END_VAR
BEGIN
END_DATA_BLOCK

DATA_BLOCK "IEC_Counter_0_DB Mauvaises"   // DB3
// stored: InstanceOfName CTU_SFB, OfSystemLibElement CTU, OfSystemLibVersion 1.0
"CTU_SFB"
   // VAR_INPUT
   //    CU : Bool;
   //    R : Bool;
   //    PV : Int;
   // END_VAR
   // VAR_OUTPUT
   //    Q : Bool;
   //    CV : Int;
   // END_VAR
   // VAR RETAIN
   //    CUO : Bool;
   // END_VAR
BEGIN
END_DATA_BLOCK

DATA_BLOCK "IEC_Counter_0_DB Noires"   // DB1
// stored: InstanceOfName CTU_SFB, OfSystemLibElement CTU, OfSystemLibVersion 1.0
"CTU_SFB"
   // VAR_INPUT
   //    CU : Bool;
   //    R : Bool;
   //    PV : Int;
   // END_VAR
   // VAR_OUTPUT
   //    Q : Bool;
   //    CV : Int;
   // END_VAR
   // VAR RETAIN
   //    CUO : Bool;
   // END_VAR
BEGIN
END_DATA_BLOCK
